{attribute 'qualified_only'}
{attribute 'strict'}
{attribute 'to_string'}
TYPE actorID_t :
(
	ACTOR_0 := 0,
	ACTOR_1,
	ACTOR_2,
	ACTOR_3,
	ACTOR_GRIPPER_RIGHT_LEFT,
	ACTOR_GRIPPER_OPEN_CLOSE,
	ACTOR_GRIPPER_UP_DOWN,
	ACTOR_Y1_OUT,
	ACTOR_Y2_OUT,
	ACTOR_Y3_OUT
);
END_TYPE

(* stored: Version 1.1.0.1
   DUT actorID_t: Id {38fea462-d6ae-4693-9b1a-7a0599fda445} *)
